% RSLogix 500 project LAB 9.RSS, saved by version 8.30.00.16 %
PROJECT "UNTITLED"    % processor: MicroLogix 1000 %

PROGRAM FILES
  LAD 2 "MAIN_PROG"  11 rungs
  LAD 3 "USER_FAULT"  1 rungs
  LAD 4 "HSC_INT"  1 rungs
  LAD 5 "STI_INT"  1 rungs
  LAD 6, 7, 8, 9, 10, 11, 12, 13, 14, 15, 16: only END

DATA FILES
  O0 OUTPUT  1 elements
  I1 INPUT  2 elements
  S2 STATUS  33 elements
  B3 BINARY  32 elements
  T4 TIMER  40 elements
  C5 COUNTER  32 elements
  R6 CONTROL  16 elements
  N7 INTEGER  105 elements

LADDER 2 "MAIN_PROG"
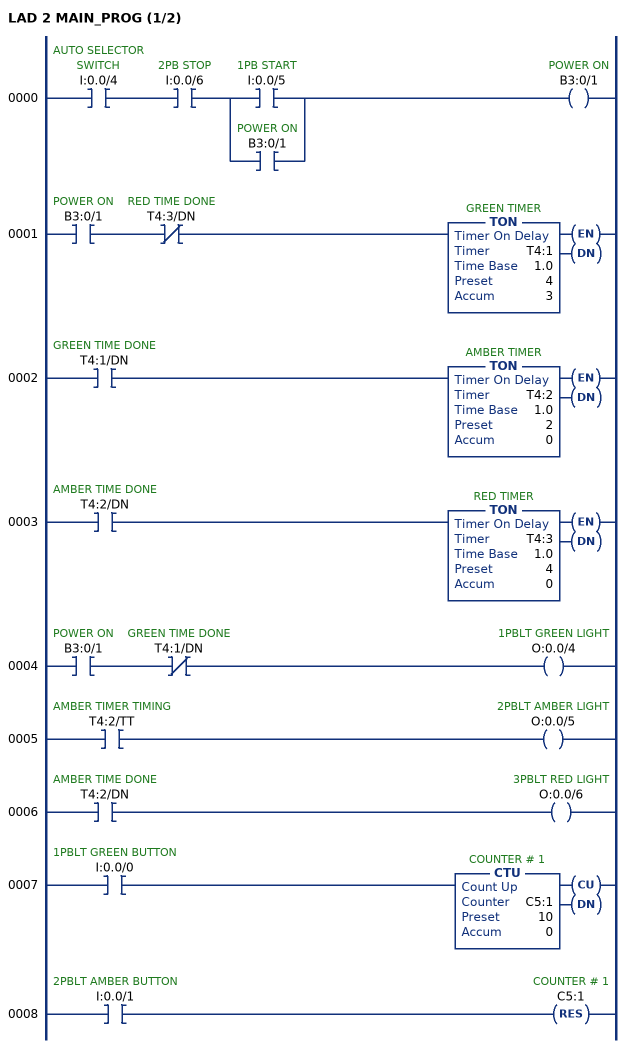
% Rung: 0 %  % edit flag set %
SOR XIC I:0.0/4 XIC I:0.0/6 BST XIC I:0.0/5 NXB XIC B3:0/1 BND OTE B3:0/1 EOR
%   I:0.0/4  "AUTO SELECTOR SWITCH" %
%   I:0.0/6  "2PB STOP" %
%   I:0.0/5  "1PB START" %
%   B3:0/1  "POWER ON" %
% Rung: 1 %  % edit flag set %
SOR XIC B3:0/1 XIO T4:3/DN TON T4:1 1.0 4 3 EOR
%   B3:0/1  "POWER ON" %
%   T4:3/DN  "RED TIME DONE" %
%   T4:1  "GREEN TIMER" %
% Rung: 2 %  % edit flag set %
SOR XIC T4:1/DN TON T4:2 1.0 2 0 EOR
%   T4:1/DN  "GREEN TIME DONE" %
%   T4:2  "AMBER TIMER" %
% Rung: 3 %  % edit flag set %
SOR XIC T4:2/DN TON T4:3 1.0 4 0 EOR
%   T4:2/DN  "AMBER TIME DONE" %
%   T4:3  "RED TIMER" %
% Rung: 4 %  % edit flag set %
SOR XIC B3:0/1 XIO T4:1/DN OTE O:0.0/4 EOR
%   B3:0/1  "POWER ON" %
%   T4:1/DN  "GREEN TIME DONE" %
%   O:0.0/4  "1PBLT GREEN LIGHT" %
% Rung: 5 %  % edit flag set %
SOR XIC T4:2/TT OTE O:0.0/5 EOR
%   T4:2/TT  "AMBER TIMER TIMING" %
%   O:0.0/5  "2PBLT AMBER LIGHT" %
% Rung: 6 %  % edit flag set %
SOR XIC T4:2/DN OTE O:0.0/6 EOR
%   T4:2/DN  "AMBER TIME DONE" %
%   O:0.0/6  "3PBLT RED LIGHT" %
% Rung: 7 %  % edit flag set %
SOR XIC I:0.0/0 CTU C5:1 10 0 EOR
%   I:0.0/0  "1PBLT GREEN BUTTON" %
%   C5:1  "COUNTER # 1" %
% Rung: 8 %  % edit flag set %
SOR XIC I:0.0/1 RES C5:1 EOR
%   I:0.0/1  "2PBLT AMBER BUTTON" %
%   C5:1  "COUNTER # 1" %

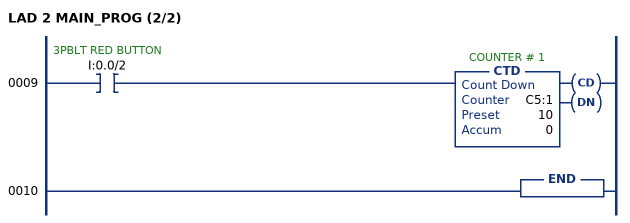
% Rung: 9 %  % edit flag set %
SOR XIC I:0.0/2 CTD C5:1 10 0 EOR
%   I:0.0/2  "3PBLT RED BUTTON" %
%   C5:1  "COUNTER # 1" %
% Rung: 10 %
SOR END EOR
